//==================================================================================================
//							Beckhoff Automation Poland
//									03.01.2023
//
// Code owner: TG
//
// Sample Interface to handle NC Axis
//
// Used libraries: 
//	Tc2_MC2								|| 3.3.48.0
//
//  v1.0	|| TC v 3.1.4024.35		|| First edition
//==================================================================================================
INTERFACE I_AxisControlBase

PROPERTY bConsequentialError 					: BOOL
GET
END_GET
END_PROPERTY

PROPERTY bDisabled 								: BOOL
GET
END_GET
END_PROPERTY

PROPERTY bDriveError 							: BOOL
GET
END_GET
END_PROPERTY

PROPERTY bEnabled 								: BOOL
GET
END_GET
END_PROPERTY

PROPERTY bEnableNegative 						: BOOL
GET
END_GET
SET
END_SET
END_PROPERTY

PROPERTY bEnablePositive 						: BOOL
GET
END_GET
SET
END_SET
END_PROPERTY

PROPERTY bError 									: BOOL
GET
END_GET
END_PROPERTY

PROPERTY bExecuteEstop 							: BOOL
GET
END_GET
SET
END_SET
END_PROPERTY

PROPERTY bLimitSwitchStateMax 					: BOOL
GET
END_GET
SET
END_SET
END_PROPERTY

PROPERTY bLimitSwitchStateMin 					: BOOL
GET
END_GET
SET
END_SET
END_PROPERTY

PROPERTY bMoving 								: BOOL
GET
END_GET
END_PROPERTY

PROPERTY bNotMoving 								: BOOL
GET
END_GET
END_PROPERTY

PROPERTY bSimulationAxis 						: BOOL
GET
END_GET
END_PROPERTY

METHOD Disable 									: BOOL
END_METHOD

PROPERTY eBufferMode 							: MC_BufferMode
GET
END_GET
SET
END_SET
END_PROPERTY

PROPERTY eDirection 								: Tc2_MC2.MC_Direction
GET
END_GET
SET
END_SET
END_PROPERTY

PROPERTY eJogMode 								: Tc2_MC2.E_JogMode
GET
END_GET
SET
END_SET
END_PROPERTY

METHOD Enable 									: BOOL
END_METHOD

METHOD EStop 									: REFERENCE TO Tc2_MC2.ST_McOutputs
VAR_INPUT
	bExecute									: BOOL;
END_VAR
END_METHOD

METHOD EStopClear 								: BOOL
END_METHOD

METHOD EStopEx 									: BOOL
END_METHOD

PROPERTY fAcceleration 							: LREAL
GET
END_GET
SET
END_SET
END_PROPERTY

PROPERTY fActAcc 								: LREAL
GET
END_GET
END_PROPERTY

PROPERTY fActPos 								: LREAL
GET
END_GET
END_PROPERTY

PROPERTY fActTorque 								: LREAL
GET
END_GET
END_PROPERTY

PROPERTY fActVelo 								: LREAL
GET
END_GET
END_PROPERTY

PROPERTY fDeceleration 							: LREAL
GET
END_GET
SET
END_SET
END_PROPERTY

PROPERTY fDecelerationEstop 						: LREAL
GET
END_GET
SET
END_SET
END_PROPERTY

PROPERTY fDistance 								: LREAL
GET
END_GET
SET
END_SET
END_PROPERTY

PROPERTY fGearRatio 								: LREAL
GET
END_GET
SET
END_SET
END_PROPERTY

PROPERTY fJerk 									: LREAL
GET
END_GET
SET
END_SET
END_PROPERTY

PROPERTY fJerkEstop 								: LREAL
GET
END_GET
SET
END_SET
END_PROPERTY

PROPERTY fLimitSwitchPositionMax 				: LREAL
GET
END_GET
SET
END_SET
END_PROPERTY

PROPERTY fLimitSwitchPositionMin 				: LREAL
GET
END_GET
SET
END_SET
END_PROPERTY

PROPERTY fOverride 								: LREAL
GET
END_GET
SET
END_SET
END_PROPERTY

PROPERTY fPosition 								: LREAL
GET
END_GET
SET
END_SET
END_PROPERTY

PROPERTY fSetAcc 								: LREAL
GET
END_GET
END_PROPERTY

PROPERTY fSetPos 								: LREAL
GET
END_GET
END_PROPERTY

PROPERTY fSetVelo 								: LREAL
GET
END_GET
END_PROPERTY

PROPERTY fVelocity 								: LREAL
GET
END_GET
SET
END_SET
END_PROPERTY

METHOD Halt 									: REFERENCE TO Tc2_MC2.ST_McOutputs
VAR_INPUT
	bExecute									: BOOL;
END_VAR
END_METHOD

METHOD HaltClear 								: BOOL
END_METHOD

METHOD HaltEx 									: BOOL
END_METHOD

METHOD Jog 										: REFERENCE TO Tc2_MC2.ST_McOutputs
VAR_INPUT
	bFw											: BOOL;
	bBw											: BOOL;
END_VAR
END_METHOD

METHOD JogBwEx 									: BOOL
END_METHOD

METHOD JogClear 								: BOOL
END_METHOD

METHOD JogContinous 							: REFERENCE TO Tc2_MC2.ST_McOutputs
VAR_INPUT
	bFw											: BOOL;
	bBw											: BOOL;
END_VAR
END_METHOD

METHOD JogFast 									: REFERENCE TO Tc2_MC2.ST_McOutputs
VAR_INPUT
	bFw											: BOOL;
	bBw											: BOOL;
END_VAR
END_METHOD

METHOD JogFwEx 									: BOOL
END_METHOD

METHOD JogInching 								: REFERENCE TO Tc2_MC2.ST_McOutputs
VAR_INPUT
	bFw											: BOOL;
	bBw											: BOOL;
END_VAR
END_METHOD

METHOD JogInchingModulo 						: REFERENCE TO Tc2_MC2.ST_McOutputs
VAR_INPUT
	bFw											: BOOL;
	bBw											: BOOL;
END_VAR
END_METHOD

METHOD JogSlow 									: REFERENCE TO Tc2_MC2.ST_McOutputs
VAR_INPUT
	bFw											: BOOL;
	bBw											: BOOL;
END_VAR
END_METHOD

METHOD LimitSwitchDisable 						: REFERENCE TO Tc2_MC2.ST_McOutputs
VAR_INPUT
	bExecute									: BOOL;
END_VAR
END_METHOD

METHOD LimitSwitchDisableMax 					: REFERENCE TO Tc2_MC2.ST_McOutputs
VAR_INPUT
	bExecute									: BOOL;
END_VAR
END_METHOD

METHOD LimitSwitchDisableMin 					: REFERENCE TO Tc2_MC2.ST_McOutputs
VAR_INPUT
	bExecute									: BOOL;
END_VAR
END_METHOD

METHOD LimitSwitchEnable 						: REFERENCE TO Tc2_MC2.ST_McOutputs
VAR_INPUT
	bExecute									: BOOL;
END_VAR
END_METHOD

METHOD LimitSwitchEnableMax 					: REFERENCE TO Tc2_MC2.ST_McOutputs
VAR_INPUT
	bExecute									: BOOL;
END_VAR
END_METHOD

METHOD LimitSwitchEnableMin 					: REFERENCE TO Tc2_MC2.ST_McOutputs
VAR_INPUT
	bExecute									: BOOL;
END_VAR
END_METHOD

METHOD LimitSwitchRead 							: REFERENCE TO Tc2_MC2.ST_McOutputs
VAR_INPUT
	bExecute									: BOOL;
END_VAR
END_METHOD

METHOD LimitSwitchWrite 						: REFERENCE TO Tc2_MC2.ST_McOutputs
VAR_INPUT
	bExecute									: BOOL;
END_VAR
END_METHOD

METHOD LimitSwitchWriteMax 						: REFERENCE TO Tc2_MC2.ST_McOutputs
VAR_INPUT
	bExecute									: BOOL;
END_VAR
END_METHOD

METHOD LimitSwitchWriteMin 						: REFERENCE TO Tc2_MC2.ST_McOutputs
VAR_INPUT
	bExecute									: BOOL;
END_VAR
END_METHOD

METHOD Manual 									: BOOL
VAR_INPUT
	stManual									: REFERENCE TO ST_AxisControlManual;
END_VAR
END_METHOD

METHOD MoveAbsolute 							: REFERENCE TO Tc2_MC2.ST_McOutputs
VAR_INPUT
	bExecute									: BOOL;
END_VAR
END_METHOD

METHOD MoveAbsolute2 							: REFERENCE TO Tc2_MC2.ST_McOutputs
VAR_INPUT
	bExecute									: BOOL;
END_VAR
END_METHOD

METHOD MoveAbsoluteClear 						: BOOL
END_METHOD

METHOD MoveAbsoluteClear2 						: BOOL
END_METHOD

METHOD MoveAbsoluteEx 							: BOOL
END_METHOD

METHOD MoveAbsoluteEx2 							: BOOL
END_METHOD

METHOD MoveModulo 								: REFERENCE TO Tc2_MC2.ST_McOutputs
VAR_INPUT
	bExecute									: BOOL;
END_VAR
END_METHOD

METHOD MoveModulo2 								: REFERENCE TO Tc2_MC2.ST_McOutputs
VAR_INPUT
	bExecute									: BOOL;
END_VAR
END_METHOD

METHOD MoveModuloClear 							: BOOL
END_METHOD

METHOD MoveModuloClear2 						: BOOL
END_METHOD

METHOD MoveModuloCurrent 						: REFERENCE TO Tc2_MC2.ST_McOutputs
VAR_INPUT
	bExecute									: BOOL;
END_VAR
END_METHOD

METHOD MoveModuloCurrent2 						: REFERENCE TO Tc2_MC2.ST_McOutputs
VAR_INPUT
	bExecute									: BOOL;
END_VAR
END_METHOD

METHOD MoveModuloEx 							: BOOL
END_METHOD

METHOD MoveModuloEx2 							: BOOL
END_METHOD

METHOD MoveModuloNeg 							: REFERENCE TO Tc2_MC2.ST_McOutputs
VAR_INPUT
	bExecute									: BOOL;
END_VAR
END_METHOD

METHOD MoveModuloNeg2 							: REFERENCE TO Tc2_MC2.ST_McOutputs
VAR_INPUT
	bExecute									: BOOL;
END_VAR
END_METHOD

METHOD MoveModuloPos 							: REFERENCE TO Tc2_MC2.ST_McOutputs
VAR_INPUT
	bExecute									: BOOL;
END_VAR
END_METHOD

METHOD MoveModuloPos2 							: REFERENCE TO Tc2_MC2.ST_McOutputs
VAR_INPUT
	bExecute									: BOOL;
END_VAR
END_METHOD

METHOD MoveModuloShort 							: REFERENCE TO Tc2_MC2.ST_McOutputs
VAR_INPUT
	bExecute									: BOOL;
END_VAR
END_METHOD

METHOD MoveModuloShort2 						: REFERENCE TO Tc2_MC2.ST_McOutputs
VAR_INPUT
	bExecute									: BOOL;
END_VAR
END_METHOD

METHOD MoveRelative 							: REFERENCE TO Tc2_MC2.ST_McOutputs
VAR_INPUT
	bExecute									: BOOL;
END_VAR
END_METHOD

METHOD MoveRelative2 							: REFERENCE TO Tc2_MC2.ST_McOutputs
VAR_INPUT
	bExecute									: BOOL;
END_VAR
END_METHOD

METHOD MoveRelativeClear 						: BOOL
END_METHOD

METHOD MoveRelativeClear2 						: BOOL
END_METHOD

METHOD MoveRelativeEx 							: BOOL
END_METHOD

METHOD MoveRelativeEx2 							: BOOL
END_METHOD

METHOD MoveVelocity 							: REFERENCE TO Tc2_MC2.ST_McOutputs
VAR_INPUT
	bExecute									: BOOL;
END_VAR
END_METHOD

METHOD MoveVelocity2 							: REFERENCE TO Tc2_MC2.ST_McOutputs
VAR_INPUT
	bExecute									: BOOL;
END_VAR
END_METHOD

METHOD MoveVelocityClear 						: BOOL
END_METHOD

METHOD MoveVelocityClear2 						: BOOL
END_METHOD

METHOD MoveVelocityEx 							: BOOL
END_METHOD

METHOD MoveVelocityEx2 							: BOOL
END_METHOD

PROPERTY nErrorId 								: UDINT
GET
END_GET
END_PROPERTY

PROPERTY pAbsolute 								: REFERENCE TO Tc2_MC2.ST_McOutputs
GET
END_GET
SET
END_SET
END_PROPERTY

PROPERTY pAbsolute2 							: REFERENCE TO Tc2_MC2.ST_McOutputs
GET
END_GET
SET
END_SET
END_PROPERTY

PROPERTY pEStop 								: REFERENCE TO Tc2_MC2.ST_McOutputs
GET
END_GET
SET
END_SET
END_PROPERTY

PROPERTY pGear 									: REFERENCE TO Tc2_MC2.ST_McOutputs
GET
END_GET
SET
END_SET
END_PROPERTY

PROPERTY pHalt 									: REFERENCE TO Tc2_MC2.ST_McOutputs
GET
END_GET
SET
END_SET
END_PROPERTY

PROPERTY pHome 									: REFERENCE TO Tc2_MC2.ST_McOutputs
GET
END_GET
SET
END_SET
END_PROPERTY

PROPERTY pJog 									: REFERENCE TO Tc2_MC2.ST_McOutputs
GET
END_GET
SET
END_SET
END_PROPERTY

PROPERTY pLimitSwitch 							: REFERENCE TO Tc2_MC2.ST_McOutputs
GET
END_GET
SET
END_SET
END_PROPERTY

PROPERTY pModulo 								: REFERENCE TO Tc2_MC2.ST_McOutputs
GET
END_GET
SET
END_SET
END_PROPERTY

PROPERTY pModulo2 								: REFERENCE TO Tc2_MC2.ST_McOutputs
GET
END_GET
SET
END_SET
END_PROPERTY

PROPERTY pOut 									: REFERENCE TO Tc2_MC2.ST_McOutputs
GET
END_GET
SET
END_SET
END_PROPERTY

METHOD Power 									: REFERENCE TO Tc2_MC2.ST_McOutputs
END_METHOD

PROPERTY pPower 								: REFERENCE TO Tc2_MC2.ST_McOutputs
GET
END_GET
SET
END_SET
END_PROPERTY

PROPERTY pRelative 								: REFERENCE TO Tc2_MC2.ST_McOutputs
GET
END_GET
SET
END_SET
END_PROPERTY

PROPERTY pRelative2 							: REFERENCE TO Tc2_MC2.ST_McOutputs
GET
END_GET
SET
END_SET
END_PROPERTY

PROPERTY pReset 								: REFERENCE TO Tc2_MC2.ST_McOutputs
GET
END_GET
SET
END_SET
END_PROPERTY

PROPERTY pSetPos 								: REFERENCE TO Tc2_MC2.ST_McOutputs
GET
END_GET
SET
END_SET
END_PROPERTY

PROPERTY pStop 									: REFERENCE TO Tc2_MC2.ST_McOutputs
GET
END_GET
SET
END_SET
END_PROPERTY

PROPERTY pVelocity 								: REFERENCE TO Tc2_MC2.ST_McOutputs
GET
END_GET
SET
END_SET
END_PROPERTY

PROPERTY pVelocity2 							: REFERENCE TO Tc2_MC2.ST_McOutputs
GET
END_GET
SET
END_SET
END_PROPERTY

METHOD Reset 									: REFERENCE TO Tc2_MC2.ST_McOutputs
VAR_INPUT
	bExecute									: BOOL;
END_VAR
END_METHOD

METHOD ResetClear 								: BOOL
END_METHOD

METHOD ResetEx 									: BOOL
END_METHOD

METHOD SetPos 									: REFERENCE TO Tc2_MC2.ST_McOutputs
VAR_INPUT
	bExecute									: BOOL;
	bMode										: BOOL;	// RELATIVE=True, ABSOLUTE=False (Default)
	stOptions									: ST_SetPositionOptions;
END_VAR
END_METHOD

METHOD SetPosClear 								: BOOL
END_METHOD

METHOD SetPosEx 								: BOOL
VAR_INPUT
	bMode										: BOOL;	// RELATIVE=True, ABSOLUTE=False (Default)
	stOptions									: ST_SetPositionOptions;
END_VAR
END_METHOD

METHOD Stop 									: REFERENCE TO Tc2_MC2.ST_McOutputs
VAR_INPUT
	bExecute									: BOOL;
END_VAR
END_METHOD

METHOD StopClear 								: BOOL
END_METHOD

METHOD StopEx 									: BOOL
END_METHOD

END_INTERFACE

(* stored: Version 1.2.0.0, ProductVersion 3.1.4026.13, FileIdentifier af8879eb0a853c8b8a2faf5f461c5a5fb7f816a5, FileSignature 846a5022d0716e9e51c4c24f1a3c1d96e25440677822c41152d35ba3f55ff7dfe35b9a56f44b0f380266457cb484493669c5fa6a710a286a14d0a15ac8002545a2e864c3b7dfc272801360d422fef2209ddc765d5d49e251fd2f96f54de76be9aaf16a6bc879804e818a3718df261a9441532c61f8b44b0a3ddeb567be3c45be34105f6d957e1a99e745a95f0d6289ce46891e9300ab5c8124c95fc33ae55e48da08ea0f5a800fb56aae621b89e4541cccfba47d82aeb91344dd453959b110db3c376fe71284f8b8af0f3ee9fc482d915a5f4dac98314140707c6af21e0c8048c8a55050c7157f15d7ce99a06070d46f3208cd7ca9f85323c412e359a0d94545
   Itf I_AxisControlBase: Id {d11b80fa-612a-4cb4-ad48-52cb78fb60b2}
   Folder Motion: Id {d130be26-7794-41b0-81e9-90f664cd3a99}
   Folder Absolute: Id {2a51fa41-381c-4e2c-aae5-55b1d99f7df0}
   Folder Jog: Id {fb9e1f04-f734-4b4c-8aac-fd3743e2187e}
   Folder Modulo: Id {23784d11-707a-4e60-a6b1-d57ba85d49b1}
   Folder Reative: Id {d193ad98-f69f-44be-8a35-3c0ff5dbbd48}
   Folder Stop: Id {b19174bb-4772-449a-826e-7044bc753940}
   Folder Velocity: Id {3fca3f0d-f55a-4eb7-a08d-bb837b2db185}
   Folder Organization: Id {bce07273-44fb-4899-8f83-a6b53db9285d}
   Folder LimitSwitch: Id {e59bc6b1-3624-421c-824a-a06137fa133a}
   Folder Power: Id {3c4f6721-43d5-426c-9c9f-452a138efe1e}
   Folder Reset: Id {788df138-80e5-4fee-b8c2-9a9f341bb42d}
   Folder SetPos: Id {02d8af2b-08cc-4046-bbe3-33fd0a30b100}
   Folder Properties: Id {e81c8c63-fb46-4298-85a3-65800c7976c7}
   Folder Commands: Id {3227cefd-2bcf-47b6-b6b3-454c4ce307a3}
   Folder FbOutputs: Id {b80820a0-c627-4227-8934-e29d60a65fc1}
   Folder Params: Id {be2dde4b-2128-4484-ae24-036a1da2f9c1}
   Folder States: Id {09e7fcd0-3168-43e5-8ca1-795b3221ff05}
   Property bConsequentialError: Id {c97f4915-3366-441c-8f43-c0a3f30fbbef}
   Get Get: Id {8ccea2ed-9706-420d-b8df-354ddf939e2b}
   Property bDisabled: Id {bf8811dd-debf-4bfb-8a66-d14dd5a5933a}
   Get Get: Id {87a5069f-9b71-4a1a-a6c3-c2d593b738af}
   Property bDriveError: Id {776557cb-87d6-4252-91a9-2b00708eaa74}
   Get Get: Id {c5559c27-c546-4deb-becd-e9da645dbba1}
   Property bEnabled: Id {135981ed-5d15-40b2-9f0e-bca4c5f445a4}
   Get Get: Id {38fca552-613d-41d3-b39e-fd38c0e27dad}
   Property bEnableNegative: Id {7ad73c49-0508-45a6-b0a4-ce68e8cf7435}
   Get Get: Id {a4da61fe-171d-49b5-be9c-a85a7874267f}
   Set Set: Id {4197796e-484e-496c-8247-d311b10b0ce0}
   Property bEnablePositive: Id {7a1f9487-d8d4-47ed-9e3a-b32eabc55906}
   Get Get: Id {c3f375a1-02db-49e3-8ec8-466d0644ac3d}
   Set Set: Id {adc90a24-fedf-4309-a943-ce15a5935ed8}
   Property bError: Id {47c627df-33aa-4067-817b-b4db0ebe2979}
   Get Get: Id {363f552e-74c7-410b-a846-da0c5cd6d778}
   Property bExecuteEstop: Id {fa87e572-ba44-401b-9c46-addc93e5a742}
   Get Get: Id {31d09694-323e-4467-99ff-3979c1d2b3d6}
   Set Set: Id {cb87e452-acec-4c59-ac0b-25a891d6642b}
   Property bLimitSwitchStateMax: Id {2a0effcf-adc1-4597-8182-b388587eaeeb}
   Get Get: Id {2ed178e4-a861-4d51-9fb7-a2cf1ed351f5}
   Set Set: Id {66fb67d8-95e7-4365-a70c-5d738eb36658}
   Property bLimitSwitchStateMin: Id {19918917-d09f-44e4-b2b7-a02967570b26}
   Get Get: Id {fbe93497-8246-46ab-a07e-7d0011282b6c}
   Set Set: Id {7aa42a05-7789-45f8-8d62-92a3b5dde084}
   Property bMoving: Id {68bfb632-b2fb-4190-a302-5230be05db6b}
   Get Get: Id {d65415d1-2257-4b92-8202-cc349426f660}
   Property bNotMoving: Id {3076d361-c3f5-49a6-98aa-8fb1a4853440}
   Get Get: Id {9ae9bde0-4197-429a-a0d8-ada45305e23f}
   Property bSimulationAxis: Id {b9218feb-dd7c-41f4-a142-b645f59cf38c}
   Get Get: Id {d30ad198-8012-462e-8ca8-7ce15b50f69c}
   Method Disable: Id {bd214242-9b96-4ccd-b949-640c2f8d5197}
   Property eBufferMode: Id {8e1844ec-75bd-48cb-83b8-91f598379793}
   Get Get: Id {f7357c5a-4000-4943-aed4-b98d6d786497}
   Set Set: Id {610645e6-e5f5-461d-a277-468cba31a129}
   Property eDirection: Id {9e58b543-211f-45d0-937c-0a7bb35c272e}
   Get Get: Id {b77f4a25-f824-442a-b427-d99408a8b1e1}
   Set Set: Id {7791030c-8820-4363-b2b8-09af88d2060f}
   Property eJogMode: Id {1e8c9ec2-5637-46cb-bb89-d20a14f3de19}
   Get Get: Id {1cee8e99-593c-41a3-8469-4f4aac0648a4}
   Set Set: Id {e78b90ed-14ef-4935-916f-456c2a1e7fc2}
   Method Enable: Id {398790f0-f56f-4ac4-a5a7-3d440e1549af}
   Method EStop: Id {c794f49d-96c5-4fc7-86a6-ce94fc6c6d4d}
   Method EStopClear: Id {9d5f12de-d8e0-40bc-b07c-3b18fb66e490}
   Method EStopEx: Id {1826c960-7fb9-4ac4-8690-2f969e642532}
   Property fAcceleration: Id {a2bda479-8a33-4374-a54c-744f014b1103}
   Get Get: Id {5d6130ac-da12-46a5-aaf6-b6a2c118021b}
   Set Set: Id {14766452-96a3-45e1-889a-5602f9d7bb7d}
   Property fActAcc: Id {02a1c01f-06a5-4f81-a73a-0cb6af253c96}
   Get Get: Id {8b27d2d2-a82a-418d-b22e-9219ded85fc0}
   Property fActPos: Id {dca6003b-9f1b-49f5-9f8c-0087b7bd8c60}
   Get Get: Id {e6268f6f-4f6c-43b8-ad15-96826b7e4566}
   Property fActTorque: Id {66e0514d-66be-4182-821a-29ba69e3dd59}
   Get Get: Id {495687e5-e3ae-4d31-b4fc-27267bca1bf9}
   Property fActVelo: Id {cd49e29c-046e-4238-84e5-aae33e7ea11f}
   Get Get: Id {304da801-85be-4871-ac85-d99daef5e25a}
   Property fDeceleration: Id {0b97fe45-52d0-4b46-a608-de5ca438b36f}
   Get Get: Id {fd81ea57-fefb-4e03-9091-322a4b961d2b}
   Set Set: Id {64b660bb-033c-4ce0-8528-6b634eaa9be4}
   Property fDecelerationEstop: Id {a64b079c-2c41-4852-aee9-da5081029c39}
   Get Get: Id {f68bbbce-38cf-4d42-9dce-fc0698e77a07}
   Set Set: Id {291376e2-f512-4974-aa0f-091199099a09}
   Property fDistance: Id {480781c3-23b5-4a0a-9dde-2ca03d70ed71}
   Get Get: Id {ebe8b573-5a1f-4101-9799-fef44c3f7486}
   Set Set: Id {b30014e1-3f64-4969-8fcd-d8fd385389f8}
   Property fGearRatio: Id {c1c73b45-e2d0-481c-9956-434e2d6e87a8}
   Get Get: Id {bc23c36d-99be-418b-9b0f-cd2122feb52a}
   Set Set: Id {fc7d1fad-a0ce-47e2-b63c-30f399bd3e0c}
   Property fJerk: Id {65e25d3d-2b72-450b-ac51-680635d5b674}
   Get Get: Id {573dd5b0-7f77-43cf-a0a6-c6ae48ce56c5}
   Set Set: Id {5a51c990-e9ac-4c2a-b063-4663756c9dd0}
   Property fJerkEstop: Id {b9576498-9e3d-44a6-adb2-c565db03838c}
   Get Get: Id {0356bf1b-eddf-42b0-b625-550271c7ec0e}
   Set Set: Id {dc6515e8-668a-45e2-853b-d03d19831cb7}
   Property fLimitSwitchPositionMax: Id {cb9eb761-b312-4652-9035-f2d1fe82a88c}
   Get Get: Id {95111b77-eaed-4e1e-969a-5274226582c9}
   Set Set: Id {c5febb7a-c09e-45b5-b46f-e1522b1a6342}
   Property fLimitSwitchPositionMin: Id {5be82102-e6c6-4091-b517-e8ab0d7e5063}
   Get Get: Id {81f2ae4f-cf2c-4521-984f-3fce097a0ccc}
   Set Set: Id {3d6c3c10-f189-492e-acfd-674a21d89a77}
   Property fOverride: Id {85f5d201-0e94-4c2c-a21c-c602d8b6160c}
   Get Get: Id {9f0b2f13-eb8e-4626-9c19-4e96b0942926}
   Set Set: Id {153c7151-5636-43fd-835a-8adaf2796611}
   Property fPosition: Id {a85fe3cc-dcd7-4de8-aece-a3663385b860}
   Get Get: Id {3004c94b-b874-4927-96d0-0c322d0d2411}
   Set Set: Id {3574ccb0-9110-4c36-bf8c-b6827135f089}
   Property fSetAcc: Id {9e673bc0-8f85-4e2b-a26c-09e50fed728c}
   Get Get: Id {811fad19-5b08-4f7f-b8cf-d50a7f9e1cf1}
   Property fSetPos: Id {78bc7258-77d3-4018-a5b7-57daeb90b978}
   Get Get: Id {54911a7c-c851-481f-aaef-b751f99f764a}
   Property fSetVelo: Id {6145d75d-b1ae-4673-8d68-d197e0a74a41}
   Get Get: Id {4d9d0a9b-f190-44ca-b659-fead8f0d350d}
   Property fVelocity: Id {bc004f10-669b-4104-8073-5a20bdd4810a}
   Get Get: Id {9263caf3-0d97-4629-a390-c0839a46eb18}
   Set Set: Id {f15dd4a7-0350-4f28-a34b-2217d21883d0}
   Method Halt: Id {3fbe0eae-d4e8-4a46-9f80-e122280a4cab}
   Method HaltClear: Id {29c12ba8-f0a2-43e6-9591-269d18c1a656}
   Method HaltEx: Id {9927e298-08f5-47e1-8b71-94bb08db78f8}
   Method Jog: Id {5da1aba7-55a6-46c4-973b-5ef954192b23}
   Method JogBwEx: Id {ff151f43-3f8f-4aaa-bf25-ec57765f9e63}
   Method JogClear: Id {1451ffd4-55dd-45db-8936-e6d9b50bdeb6}
   Method JogContinous: Id {10d55127-2dc6-4bb2-8363-7f7d80883868}
   Method JogFast: Id {76ac07fe-a606-404c-8367-440779f857c0}
   Method JogFwEx: Id {781bc37e-88a2-4e31-8d8c-09920cd619d5}
   Method JogInching: Id {d7a20420-08b6-4baf-8953-d026fad3d6a9}
   Method JogInchingModulo: Id {eeda6911-9d30-40f7-82e2-dfd85929c869}
   Method JogSlow: Id {863a25bd-7295-4a2d-be6a-4fbe3055c929}
   Method LimitSwitchDisable: Id {a367468c-dc66-45d0-a8c2-e488b4e5b85c}
   Method LimitSwitchDisableMax: Id {2d83f373-a82f-4672-b7a9-aee7d80a74ce}
   Method LimitSwitchDisableMin: Id {0922a92a-87fb-4fc8-ae5b-b5443d9c4764}
   Method LimitSwitchEnable: Id {ae0932b7-1c1d-4ca4-b278-301ff18abe00}
   Method LimitSwitchEnableMax: Id {b6b5c891-50dc-49c4-ad31-e21733e172a7}
   Method LimitSwitchEnableMin: Id {ea6447cb-a1eb-459a-9a9d-52296d23ad53}
   Method LimitSwitchRead: Id {a240892a-a7d9-463d-94c9-b685c19ba4f0}
   Method LimitSwitchWrite: Id {9f75efea-98fc-4adc-b520-da1c189021f2}
   Method LimitSwitchWriteMax: Id {33aad30c-ba94-45c2-b95b-2aeade74b856}
   Method LimitSwitchWriteMin: Id {b89cce14-2107-4b53-91be-68552c0f09da}
   Method Manual: Id {1095ded9-595f-4110-95cf-19886ab6004c}
   Method MoveAbsolute: Id {9d2c27ab-aacc-4074-8691-9427efa22e07}
   Method MoveAbsolute2: Id {2923e778-ad9c-4689-a2c9-345bd2cf8232}
   Method MoveAbsoluteClear: Id {d4a81a9e-8d80-4df8-b4ca-256dbdfbf3a9}
   Method MoveAbsoluteClear2: Id {f58e3c05-f564-40f7-8ab5-909bee13387a}
   Method MoveAbsoluteEx: Id {c34a2b1c-2f60-4853-b251-b7e21464e7d6}
   Method MoveAbsoluteEx2: Id {2ab87e39-1c7c-4067-a883-649b68ef06ee}
   Method MoveModulo: Id {aa24813e-71a6-4390-865a-b5a21709324a}
   Method MoveModulo2: Id {5d6bbe30-5cd6-420e-857e-2cc649daea8d}
   Method MoveModuloClear: Id {4ed2c9d4-d0fb-4dd0-8d98-48b0f6fc9beb}
   Method MoveModuloClear2: Id {53fdd2a6-63f8-47d5-ba47-2ebf019a818d}
   Method MoveModuloCurrent: Id {c396f4b6-6faf-4a2d-9b82-7ef75e6478cb}
   Method MoveModuloCurrent2: Id {d7c3f114-e3dc-48c0-b453-ef17a74259d7}
   Method MoveModuloEx: Id {9ee8909d-fc66-433d-866e-61eca9467d6b}
   Method MoveModuloEx2: Id {f95fff8f-6c70-4a3f-8586-971022dec39e}
   Method MoveModuloNeg: Id {dd6ed9c9-12f0-4cdf-ba4f-39f43d99f95d}
   Method MoveModuloNeg2: Id {d334a3ba-b57a-4f00-bd3e-e0846d61a055}
   Method MoveModuloPos: Id {41c11b63-c707-4fb4-a638-9ddf0ba68a6f}
   Method MoveModuloPos2: Id {93d92e74-7444-43de-8bb2-f06bdb75815c}
   Method MoveModuloShort: Id {cea676f3-6448-479d-9169-f5af0e24ee70}
   Method MoveModuloShort2: Id {c36d718d-54c9-41bd-a29c-937f87855f5c}
   Method MoveRelative: Id {b3a6db8a-b279-4058-beac-0b061045d534}
   Method MoveRelative2: Id {a0c93048-b798-4897-b842-a75a11a06046}
   Method MoveRelativeClear: Id {edfc0ff9-3836-4b14-a0e3-d06d2ceac760}
   Method MoveRelativeClear2: Id {700c81e5-b00b-4887-b9d5-60231dadefec}
   Method MoveRelativeEx: Id {bb2de365-59f4-4ef3-b33f-665ecc57b561}
   Method MoveRelativeEx2: Id {e0204687-9957-4ef2-abcd-35f8b1f9c97e}
   Method MoveVelocity: Id {9b4af583-de66-472a-ad00-acec00b7d1b1}
   Method MoveVelocity2: Id {cb9a87ad-c626-4a2f-ba42-b12022907839}
   Method MoveVelocityClear: Id {f4d189cb-d580-4f1a-a0d9-f2eabad463c0}
   Method MoveVelocityClear2: Id {fa137635-cc29-4bbb-8073-fc96f95d8e0b}
   Method MoveVelocityEx: Id {2e7d607f-4ce1-4be4-bc6c-ae1e65f02447}
   Method MoveVelocityEx2: Id {3b16d586-585e-4a09-9781-42a08cebc7db}
   Property nErrorId: Id {184ca83a-4e13-4815-83c5-e577b9aa9f87}
   Get Get: Id {96f66a15-0d36-4b8a-adee-250d20ac8896}
   Property pAbsolute: Id {1e2e9374-565b-4834-9bd4-015630c956bf}
   Get Get: Id {2338b3a4-83c9-460c-a550-a1fe4036b89b}
   Set Set: Id {0de600d5-b5a4-4778-8e23-0955c0acfe5e}
   Property pAbsolute2: Id {5eda6cc2-95ac-424c-9bb4-ffca069c10cf}
   Get Get: Id {3fc9d0be-ec9d-47b8-9846-c75e015ee4e8}
   Set Set: Id {0094d29e-07fa-48e8-9fbd-5a46a79295ae}
   Property pEStop: Id {f12d172b-74a0-461a-a4b7-ce4a9026c013}
   Get Get: Id {eeace96a-0b23-4253-a0d1-ee72f8740f31}
   Set Set: Id {8dde24e5-5602-4015-969c-d332385d3738}
   Property pGear: Id {9fc71e22-65b9-4c08-9aa5-7fe5b28c87d3}
   Get Get: Id {5702b68f-7a35-4152-8136-7c758331af6f}
   Set Set: Id {ae8877b4-8e0a-4bef-ab99-4c414c97ddc3}
   Property pHalt: Id {7d6d3714-d5cc-4386-a006-21d91778460b}
   Get Get: Id {484da0cb-fb81-41af-8f2e-c30fceec6f65}
   Set Set: Id {8cb56134-fbc0-42d5-b9f3-268ebba8feb1}
   Property pHome: Id {65fda452-a1e3-40af-92bf-2d573c3b963e}
   Get Get: Id {917d6b85-8bf3-4738-b271-e8608612a545}
   Set Set: Id {9da1d874-bd84-4506-a8bf-401b3f403daa}
   Property pJog: Id {8ebbc0a8-36ae-4013-986e-50128751cdd2}
   Get Get: Id {90d01125-37aa-4192-880b-557520491df2}
   Set Set: Id {9dc97b65-58e1-4234-8d6b-0de57f9a47fd}
   Property pLimitSwitch: Id {a217ceee-d688-44b3-9835-740566f07a4d}
   Get Get: Id {e940f10e-9af5-4ee9-9463-9bc21c097828}
   Set Set: Id {1049ccf3-0b67-4f1a-84ba-a6596b4462bc}
   Property pModulo: Id {d5283824-786b-43d2-a65b-60413b9a2bc7}
   Get Get: Id {beb06278-da61-4334-9cbd-f785ee40f293}
   Set Set: Id {3dc469da-b747-48de-b058-eee95eba5dcc}
   Property pModulo2: Id {54d296f4-93f6-4a15-b535-59079b0a41d8}
   Get Get: Id {fa258a9c-fb8d-4f70-9640-d1a7dce05b59}
   Set Set: Id {bf618cdd-67a8-499b-8b5c-a10bad33fe67}
   Property pOut: Id {1f195b33-c015-494e-ab4c-b00dade95468}
   Get Get: Id {5fee0ebc-6518-4bfb-8a10-d7913f870d03}
   Set Set: Id {3bf20457-f7ba-4bff-b2aa-411ad2e5f058}
   Method Power: Id {85f58394-721c-4384-a204-0006828ce77b}
   Property pPower: Id {132ca0c5-99e6-4076-bd60-6619d1c21131}
   Get Get: Id {dc13fd2e-2f5b-4bf4-b315-58a84736d9e0}
   Set Set: Id {d2e12e16-b7db-4515-b63f-1cba868f18eb}
   Property pRelative: Id {80b518e5-e8f4-48ab-85c6-a6ffd2aab012}
   Get Get: Id {f5f47d32-0f17-4f93-9d57-f24b33336d63}
   Set Set: Id {996a1071-6e26-4e77-9d1e-8a3fb0bd7300}
   Property pRelative2: Id {349c42e6-f75d-4455-b77b-124d9f1a6cae}
   Get Get: Id {a5a2e246-2548-46dd-8f14-2dac111e6cf5}
   Set Set: Id {6ec7d1d8-2356-4811-845c-c6312d2a970f}
   Property pReset: Id {23433aa2-40b5-41a2-91a7-99744657db71}
   Get Get: Id {6637f1ed-9890-4b61-80c0-8b08b6a900d0}
   Set Set: Id {fae15d7a-bbe7-4f40-b53b-8a5bb896b9e5}
   Property pSetPos: Id {b80ce97d-71d8-4a8d-bbe6-41da38e6374c}
   Get Get: Id {de3964df-fca7-4648-a18b-187d3a34360c}
   Set Set: Id {055ed2cb-4444-44e8-94b3-a51727c11170}
   Property pStop: Id {4b067607-936c-483e-92f8-ede82db9fd85}
   Get Get: Id {e6b48a76-c017-417a-b9ed-babc698d7e4b}
   Set Set: Id {1b63a7ca-d3b7-487d-bb14-691300e5816d}
   Property pVelocity: Id {ff5ba6db-7b95-4b7d-9d1b-dbf24a500e38}
   Get Get: Id {ad36e0ad-6265-4cf5-961a-9079d6e08799}
   Set Set: Id {d629ffde-9b5f-4cdb-bdf2-347016f95630}
   Property pVelocity2: Id {878924dc-50a2-41d6-946b-caff3f462928}
   Get Get: Id {13287e6f-bb79-4690-a0dc-deb87d2a4487}
   Set Set: Id {455549d3-b3da-442a-a76c-f9f702569e01}
   Method Reset: Id {a3b59802-a1f1-4529-bce8-858537b8dcb0}
   Method ResetClear: Id {b76d7db8-f9a8-4445-9126-0c3003955195}
   Method ResetEx: Id {358f6372-93a0-4536-9546-b7677a4efe62}
   Method SetPos: Id {f706de9d-1207-4709-8c04-df0f5cdceb4c}
   Method SetPosClear: Id {f1894d08-3121-45e4-ad7e-61fcd3477621}
   Method SetPosEx: Id {c1c78259-5936-414d-b364-496543ea968b}
   Method Stop: Id {80ba87a4-ea38-405d-990f-f1e5fc485e3d}
   Method StopClear: Id {bd4e3543-1d70-43de-b633-eaaf2e85b58b}
   Method StopEx: Id {98454967-857f-4379-9650-98198d5e4014} *)
